TYPE CmpConvMerge :		//Version 02 - 06/17/2022
STRUCT
	Framework: Framework;
	MainHeartbeatOK: BOOL;
	MainConvRunning: BOOL;
	MainInAuto: BOOL;
	SpurHeartbeatOK: BOOL;
	SpurConvRunning: BOOL;
	SpurInAuto: BOOL;
	BufferFull: BOOL;
	StatusInCycleAuto: BOOL;
	FreeRunCycleStop: BOOL;
	TrafficControlMainAvailable: BOOL;
	TrafficControlMainRelease: BOOL;
	TrafficControlSpurAvailable: BOOL;
	TrafficControlSpurRelease: BOOL;
	Config: CmpConvMergeConfig;
END_STRUCT
END_TYPE

(* stored: Version 1.1.0.1, ProductVersion 3.1.4024.6
   DUT CmpConvMerge: Id {493bb9e2-29c7-4b4c-8198-8aa522654fe2} *)
